// TwinCAT 3 PLC project GantryTest
// ProgramVersion: 3.1.4020.4
// libraries:
//   Tc2_MC2, * (Beckhoff Automation GmbH)
//   Tc2_Standard, * (Beckhoff Automation GmbH)
//   Tc2_System, * (Beckhoff Automation GmbH)
//   Tc3_Module, * (Beckhoff Automation GmbH)
// project tree:
//   / PlcTask.TcTTO
//   POUs/ MAIN.TcPOU
// real-time tasks:
//   TASK PlcTask: cycle T#10ms, priority 20, ADS port 350
// motion (NC):
//   TASK NC-Task 1 SAF: cycle T#2ms, priority 4, ADS port 501
//   TASK NC-Task 1 SVB: cycle T#10ms, priority 8, ADS port 511
//   AXIS Axis 1 (id 1)
//     Dynamic: DelayTime=0.008
//     Velo: RefSearch=0.1, RefSync=0.1, SlowManual=0.25, FastManual=0.5, Maximum=1
//     PositionAreaControl: Range=0.1
//     TargetPosControl: Range=0.1
//     OtherSettings: AllowMotionCmdToSlave=true, PulseDistancePos=0.1, PulseDistanceNeg=0.1
//     encoder EncType=29
//       EncPara: ScaleFactorNumerator=1e-06, MaxCount=#xffffffff, ReferenceSystem=1
//         Inc: RefSoftSyncMask=#x0000ffff
//     drive DrvType=24
//       Analog: VeloReferenz=1.2206875
//       TimeComp: TaskDelayCycles=1
//     controller CtrType=2
//       CtrPara: PriorControlFactor=1
//         PosDiffControl: Range=0.1
//         PID: PosKp=10, PosExtKp=1
//         Observer: BandWidth=20
//   AXIS Axis 2 (id 2)
//     Dynamic: DelayTime=0.008
//     Velo: RefSearch=0.1, RefSync=0.1, SlowManual=0.25, FastManual=0.5, Maximum=0.1
//     PositionAreaControl: Range=0.1
//     TargetPosControl: Range=0.1
//     OtherSettings: AllowMotionCmdToSlave=true, PulseDistancePos=0.1, PulseDistanceNeg=0.1
//     encoder EncType=29
//       EncPara: ScaleFactorNumerator=1e-06, MaxCount=#xffffffff, ReferenceSystem=1
//         Inc: RefSoftSyncMask=#x0000ffff
//     drive DrvType=24
//       DrvPara: Inverse=true
//         Analog: VeloReferenz=1.2206875
//         TimeComp: TaskDelayCycles=1
//     controller CtrType=2
//       CtrPara: PriorControlFactor=1
//         PosDiffControl: Range=0.1
//         PID: PosKp=10, PosExtKp=1
//         Observer: BandWidth=20
// I/O:
//   DEVICE Device 1 (EtherCAT), AmsNetId 5.59.121.62.2.1
//     Term 1 (EK1200) [EK1200-5000 EtherCAT Power supply (2A E-Bus)]
//       Term 2 (EL7041-1000) [EL7041-1000 1Ch. Stepper motor output stage (50V, 5A, standard)]
//       Term 3 (EL7041-1000) [EL7041-1000 1Ch. Stepper motor output stage (50V, 5A, standard)]
//       Term 4 (EL5042) [EL5042 2Ch. BiSS-C Encoder]
//       Term 5 (EL1004) [EL1004 4Ch. Dig. Input 24V, 3ms]
//       Term 6 (EL9011) [EL9011 End Terminal]
// variable links:
//   (this object) <-> Device 1 (EtherCAT)/Term 1 (EK1200)/Term 2 (EL7041-1000)
//     Drive/Inputs/In/nState1 @bit 3 <-> STM Status/Status/Error
//     Drive/Inputs/In/nState1 @bit 5 <-> STM Status/Status/Moving negative
//     Drive/Inputs/In/nState1 @bit 4 <-> STM Status/Status/Moving positive
//     Drive/Inputs/In/nState1 @bit 1 <-> STM Status/Status/Ready
//     Drive/Inputs/In/nState1 <-> STM Status/Status/Ready to enable
//     Drive/Inputs/In/nState1 @bit 6 <-> STM Status/Status/Torque reduced
//     Drive/Inputs/In/nState1 @bit 2 <-> STM Status/Status/Warning
//     Drive/Inputs/In/nState2 @bit 3 <-> STM Status/Status/Digital input 1
//     Drive/Inputs/In/nState2 @bit 4 <-> STM Status/Status/Digital input 2
//     Drive/Inputs/In/nState2 @bit 5 <-> STM Status/Status/Sync error
//     Drive/Inputs/In/nState2 @bit 7 <-> STM Status/Status/TxPDO Toggle
//     Drive/Inputs/In/nState4 @bit 1 <-> WcState/InputToggle
//     Drive/Inputs/In/nState4 <-> WcState/WcState
//     Drive/Outputs/Out/nCtrl1 <-> STM Control/Control/Enable
//     Drive/Outputs/Out/nCtrl1 @bit 2 <-> STM Control/Control/Reduce torque
//     Drive/Outputs/Out/nCtrl1 @bit 1 <-> STM Control/Control/Reset
//     Drive/Outputs/Out/nDataOut2[0] <-> STM Velocity/Velocity
//   (this object) <-> Device 1 (EtherCAT)/Term 1 (EK1200)/Term 4 (EL5042)
//     Enc/Inputs/In/nComState @bit 1 <-> WcState/InputToggle
//     Enc/Inputs/In/nComState <-> WcState/WcState
//     Enc/Inputs/In/nDataIn1 <-> FB Inputs Channel 1/Position
//     Enc/Inputs/In/nDataIn1 <-> FB Inputs Channel 2/Position
//     Enc/Inputs/In/nState1 @bit 12 <-> FB Inputs Channel 1/Status/Diag
//     Enc/Inputs/In/nState1 @bit 12 <-> FB Inputs Channel 2/Status/Diag
//     Enc/Inputs/In/nState1 @bit 1 <-> FB Inputs Channel 1/Status/Error
//     Enc/Inputs/In/nState1 @bit 1 <-> FB Inputs Channel 2/Status/Error
//     Enc/Inputs/In/nState1 @bit 14 <-> FB Inputs Channel 1/Status/Input cycle counter
//     Enc/Inputs/In/nState1 @bit 14 <-> FB Inputs Channel 2/Status/Input cycle counter
//     Enc/Inputs/In/nState1 @bit 2 <-> FB Inputs Channel 1/Status/Ready
//     Enc/Inputs/In/nState1 @bit 2 <-> FB Inputs Channel 2/Status/Ready
//     Enc/Inputs/In/nState1 @bit 13 <-> FB Inputs Channel 1/Status/TxPDO State
//     Enc/Inputs/In/nState1 @bit 13 <-> FB Inputs Channel 2/Status/TxPDO State
//     Enc/Inputs/In/nState1 <-> FB Inputs Channel 1/Status/Warning
//     Enc/Inputs/In/nState1 <-> FB Inputs Channel 2/Status/Warning
//   (this object) <-> Device 1 (EtherCAT)/Term 1 (EK1200)/Term 3 (EL7041-1000)
//     Drive/Inputs/In/nState1 @bit 3 <-> STM Status/Status/Error
//     Drive/Inputs/In/nState1 @bit 5 <-> STM Status/Status/Moving negative
//     Drive/Inputs/In/nState1 @bit 4 <-> STM Status/Status/Moving positive
//     Drive/Inputs/In/nState1 @bit 1 <-> STM Status/Status/Ready
//     Drive/Inputs/In/nState1 <-> STM Status/Status/Ready to enable
//     Drive/Inputs/In/nState1 @bit 6 <-> STM Status/Status/Torque reduced
//     Drive/Inputs/In/nState1 @bit 2 <-> STM Status/Status/Warning
//     Drive/Inputs/In/nState2 @bit 3 <-> STM Status/Status/Digital input 1
//     Drive/Inputs/In/nState2 @bit 4 <-> STM Status/Status/Digital input 2
//     Drive/Inputs/In/nState2 @bit 5 <-> STM Status/Status/Sync error
//     Drive/Inputs/In/nState2 @bit 7 <-> STM Status/Status/TxPDO Toggle
//     Drive/Inputs/In/nState4 @bit 1 <-> WcState/InputToggle
//     Drive/Inputs/In/nState4 <-> WcState/WcState
//     Drive/Outputs/Out/nCtrl1 <-> STM Control/Control/Enable
//     Drive/Outputs/Out/nCtrl1 @bit 2 <-> STM Control/Control/Reduce torque
//     Drive/Outputs/Out/nCtrl1 @bit 1 <-> STM Control/Control/Reset
//     Drive/Outputs/Out/nDataOut2[0] <-> STM Velocity/Velocity
//   GantryTest Instance <-> Device 1 (EtherCAT)/Term 1 (EK1200)/Term 2 (EL7041-1000)
//     PlcTask Inputs/MAIN.bLimBwd1 <-> STM Status/Status/Digital input 2
//     PlcTask Inputs/MAIN.bLimFwd1 <-> STM Status/Status/Digital input 1
//   GantryTest Instance <-> Device 1 (EtherCAT)/Term 1 (EK1200)/Term 3 (EL7041-1000)
//     PlcTask Inputs/MAIN.bLimBwd2 <-> STM Status/Status/Digital input 2
//     PlcTask Inputs/MAIN.bLimFwd2 <-> STM Status/Status/Digital input 1
//   GantryTest Instance <-> Device 1 (EtherCAT)/Term 1 (EK1200)/Term 4 (EL5042)
//     PlcTask Inputs/MAIN.nRawEnc1 <-> FB Inputs Channel 1/Position
//     PlcTask Inputs/MAIN.nRawEnc2 <-> FB Inputs Channel 2/Position
//   GantryTest Instance <-> Device 1 (EtherCAT)/Term 1 (EK1200)/Term 5 (EL1004)
//     PlcTask Inputs/MAIN.bSTO1 <-> Channel 1/Input
//     PlcTask Inputs/MAIN.bSTO2 <-> Channel 2/Input
//   GantryTest Instance <-> NC-Task 1 SAF/Axes/Axis 1
//     PlcTask Inputs/MAIN.Axis1.NcToPlc <-> Outputs/ToPlc
//     PlcTask Outputs/MAIN.Axis1.PlcToNc <-> Inputs/FromPlc
//   GantryTest Instance <-> NC-Task 1 SAF/Axes/Axis 2
//     PlcTask Inputs/MAIN.Axis2.NcToPlc <-> Outputs/ToPlc
//     PlcTask Outputs/MAIN.Axis2.PlcToNc <-> Inputs/FromPlc

CONFIGURATION GantryTest
    RESOURCE PLC ON TwinCAT3
        TASK PlcTask(INTERVAL := T#10ms, PRIORITY := 20);
        PROGRAM MAIN WITH PlcTask : MAIN;
    END_RESOURCE
END_CONFIGURATION

// ---- POUs/MAIN.TcPOU
PROGRAM MAIN
VAR
	Axis1: AXIS_REF;
	bEna1: BOOL;
	bEna2: BOOL;
	bSTO1 AT %I*: BOOL;
	bSTO2 AT %I*: BOOL;
	fbPower1: MC_POWER;
	bLimFwd1 AT %I*: BOOL;
	bLimBwd1 AT %I*: BOOL;
	Axis2: AXIS_REF;
	fbPower2: MC_POWER;
	bLimFwd2 AT %I*: BOOL;
	bLimBwd2 AT %I*: BOOL;
	nRawEnc1 AT %I*: ULINT;
	nRawEnc2 AT %I*: ULINT;
	nGantryOffset: LINT;
	nGantryErr: LINT;
	nAbsGantryErr: ULINT;
END_VAR

fbPower1(Axis:=Axis1,
	Enable:=bSTO1 AND bSTO2 AND bEna1,
	Enable_Positive:=bLimFwd1,
	Enable_Negative:=bLimBwd1);
fbPower2(Axis:=Axis2,
	Enable:=bSTO1 AND bSTO2 AND bEna2,
	Enable_Positive:=bLimFwd2,
	Enable_Negative:=bLimBwd2);
nGantryErr := nRawEnc2 - nRawEnc1 + nGantryOffset;
nAbsGantryErr := ABS(nGantryErr);

END_PROGRAM
